{attribute addProperty BoxType "EL3773-0000-0016"}
{attribute addProperty Id "StartTimeNextLatchAT %I*ULINT648"}
{attribute addProperty CRC "1335715474"}
{attribute addProperty SizeInBites "64"}
{attribute addProperty SizeInBytes "8"}
TYPE AI_Timestamp_NextSync1Time_4F9D6692 :
STRUCT
	{attribute addProperty Name "StartTimeNextLatch"}
	StartTimeNextLatch AT %I* : ULINT;
END_STRUCT
END_TYPE

(* stored: Version 1.2.0.0, ProductVersion 3.1.4024.9
   DUT AI_Timestamp_NextSync1Time_4F9D6692: Id {b02c9f16-7abd-49a9-9d63-efae7f0411b4} *)
